TYPE Parameter_Lokal :
STRUCT
	
	Name				:STRING(32);
	Value				:TIME;
	
END_STRUCT
END_TYPE

(* stored: Version 1.1.0.1, ProductVersion 3.1.4024.12
   DUT Parameter_Lokal: Id {55241cb6-de31-4172-bac3-4fc2e30488b2} *)
